(*
SPDX-FileCopyrightText: Â© 2026 Oleksandr Tiutyk <trofimich@gmail.com>
SPDX-License-Identifier: MIT
License: https://opensource.org/license/mit
*)

(*!
<summary>Range converter with static limits passed at construction and stored in internal fields.</summary>
<description>
Safely preserves configured limits across TwinCAT online change cycles by guarding against bInCopyCode zeroing.
</description>
*)

{attribute 'no_explicit_call' := 'do not call this function block directly'}
FUNCTION_BLOCK StaticRangeAnalogValueConverter EXTENDS AbstractRangeAnalogValueConverter
VAR_STAT
	{attribute 'hide'} 
	_ClassName : STRING := __POUNAME();
END_VAR
VAR
	{attribute 'hide'} 
	_MinAnalogValueVariable : LREAL;
	{attribute 'hide'} 
	_MaxAnalogValueVariable : LREAL;
	{attribute 'hide'} 
	_MinRawValueVariable : RAW_ANALOG_VALUE;
	{attribute 'hide'} 
	_MaxRawValueVariable : RAW_ANALOG_VALUE;
END_VAR

(*!
<summary>Gets the class name of the converter.</summary>
*)
{attribute 'monitoring' := 'call'}
PROPERTY ClassName : REFERENCE TO STRING
GET
ClassName REF= _ClassName;
END_GET
END_PROPERTY

(*!
<summary>Initializes static limits and binds internal references.</summary>
<param name="bInitRetains">TRUE: retain variables are initialized.</param>
<param name="bInCopyCode">TRUE: instance copied to copy code (online change).</param>
<param name="minAnalogValue">Minimum engineering unit value.</param>
<param name="maxAnalogValue">Maximum engineering unit value.</param>
<param name="minRawValue">Minimum raw hardware process value.</param>
<param name="maxRawValue">Maximum raw hardware process value.</param>
*)
METHOD FB_init : BOOL
VAR_INPUT
	bInitRetains : BOOL; // TRUE: the retain variables are initialized (reset warm / reset cold)
	bInCopyCode : BOOL;  // TRUE: the instance will be copied to the copy code afterward (online change)
	minAnalogValue : LREAL;
	maxAnalogValue : LREAL;
	minRawValue : RAW_ANALOG_VALUE;
	maxRawValue : RAW_ANALOG_VALUE;
END_VAR
IF NOT bInCopyCode THEN
	_MinAnalogValueVariable := minAnalogValue;
	_MaxAnalogValueVariable := maxAnalogValue;
	_MinRawValueVariable := minRawValue;
	_MaxRawValueVariable := maxRawValue;
END_IF

_MinAnalogValue REF= _MinAnalogValueVariable;
_MaxAnalogValue REF= _MaxAnalogValueVariable;
_MinRawValue REF= _MinRawValueVariable;
_MaxRawValue REF= _MaxRawValueVariable;
END_METHOD

(*!
<summary>Gets the memory size of the instance.</summary>
*)
{attribute 'monitoring' := 'call'}
PROPERTY SelfSize : ULINT
GET
SelfSize := XSIZEOF(THIS^);
END_GET
END_PROPERTY

END_FUNCTION_BLOCK

(* stored: Version 1.1.0.1
   POU StaticRangeAnalogValueConverter: Id {8bfb79ca-38fb-48e6-8fa5-f03902a6c98a}, SpecialFunc None
   Property ClassName: Id {f225b4c3-3770-4526-8d24-8f9b17c94ac6}
   Get Get: Id {1e40a6f5-8aab-44ae-954a-cfc944f55260}
   Method FB_init: Id {c27e589d-53ab-4bd9-9238-65b8df322868}
   Property SelfSize: Id {e456092c-27c0-422b-8aba-c37187fdfff9}
   Get Get: Id {373d6d1f-2cdd-4f48-96df-937f2f5a9b85} *)
